FUNCTION_BLOCK FB_TM1K2
(*
    Function block for Arrival Time Monitor (ATM) controls:
    - X, Y motion
    - Y target states
    - thermocouple

    For TM1K2, we make the following adjustments:
    - Add stTarget6 to the inputs
    - Change the array pragma from 1..6 to 1..7 (1 out and 6 in states, up from 5 in states)
    - Use E_TM1K2_States instead of E_ATM_States
	
	Add array to 1..9
*)
VAR_IN_OUT
    // Y motor (state select).
    stYStage: ST_MotionStage;
    // X motor (align target to beam).
    stXStage: ST_MotionStage;
    // The fast fault output to fault to.
    fbFFHWO: FB_HardwareFFOutput;
    // The arbiter to request beam conditions from.
    fbArbiter: FB_Arbiter;
END_VAR
VAR_INPUT
    // Settings for the OUT state.
    stOut: ST_PositionState;
    // Settings for the TARGET1 state.
    stTarget1: ST_PositionState;
    // Settings for the TARGET2 state.
    stTarget2: ST_PositionState;
    // Settings for the TARGET3 state.
    stTarget3: ST_PositionState;
    // Settings for the TARGET4 state.
    stTarget4: ST_PositionState;
    // Settings for the TARGET5 state.
    stTarget5: ST_PositionState;
    // Settings for the TARGET6 state.
    stTarget6: ST_PositionState;
    // Settings for the TARGET7 state.
    stTarget7: ST_PositionState;
    // Settings for the TARGET8 state.
    stTarget8: ST_PositionState;
    // Set this to a non-unknown value to request a new move.
    {attribute 'pytmc' := '
        pv: MMS:STATE:SET
        io: io
    '}
    eEnumSet: E_TM1K2_States;
    // Set this to TRUE to enable input state moves, or FALSE to disable them.
    bEnableMotion: BOOL;
    // Set this to TRUE to enable beam parameter checks, or FALSE to disable them.
    bEnableBeamParams: BOOL;
    // Set this to TRUE to enable position limit checks, or FALSE to disable them.
    bEnablePositionLimits: BOOL;
    // The name of the device for use in the PMPS DB lookup and diagnostic screens.
    sDeviceName: STRING;
    // The name of the transition state in the PMPS database.
    sTransitionKey: STRING;
    // Set this to TRUE to re-read the loaded database immediately (useful for debug).
    bReadDBNow: BOOL;
END_VAR
VAR_OUTPUT
    // The current position state as an enum.
    {attribute 'pytmc' := '
        pv: MMS:STATE:GET
        io: i
    '}
    eEnumGet: E_TM1K2_States;
    // The PMPS database lookup associated with the current position state.
    stDbStateParams: ST_DbStateParams;
END_VAR
VAR
    bInit: BOOL;

    fbYStage: FB_MotionStage;
    fbXStage: FB_MotionStage;

    fbStateDefaults: FB_PositionState_Defaults;

    {attribute 'pytmc' := '
        pv: MMS
        astPositionState.array: 1..7
    '}
    fbStates: FB_PositionStatePMPS1D;
    astPositionState: ARRAY[1..GeneralConstants.MAX_STATES] OF ST_PositionState;
    fbArrCheckWrite: FB_CheckPositionStateWrite;

    {attribute 'pytmc' := 'pv: STC:01'}
    fbThermoCouple1: FB_TempSensor;

    {attribute 'pytmc' :='pv: FWM'}
    fbFlowMeter: FB_AnalogInput := (iTermBits:=15, fTermMax:=60, fTermMin:=0);
END_VAR
VAR CONSTANT
    // State defaults if not provided
    fDelta: LREAL := 2;
    fAccel: LREAL := 200;
    fOutDecel: LREAL := 25;
END_VAR


IF NOT bInit THEN
    bInit := TRUE;

    stYStage.nEnableMode := E_StageEnableMode.DURING_MOTION;
    stXStage.nEnableMode := E_StageEnableMode.DURING_MOTION;

    // Partial backcompat, this used to set fVelocity too but this should be set per install
    fbStateDefaults(stPositionState:=stOut, sNameDefault:='OUT', fDeltaDefault:=fDelta, fAccelDefault:=fAccel, fDecelDefault:=fOutDecel);
    fbStateDefaults(stPositionState:=stTarget1, sNameDefault:='TARGET1', fDeltaDefault:=fDelta, fAccelDefault:=fAccel, fDecelDefault:=fAccel);
    fbStateDefaults(stPositionState:=stTarget2, sNameDefault:='TARGET2', fDeltaDefault:=fDelta, fAccelDefault:=fAccel, fDecelDefault:=fAccel);
    fbStateDefaults(stPositionState:=stTarget3, sNameDefault:='TARGET3', fDeltaDefault:=fDelta, fAccelDefault:=fAccel, fDecelDefault:=fAccel);
    fbStateDefaults(stPositionState:=stTarget4, sNameDefault:='TARGET4', fDeltaDefault:=fDelta, fAccelDefault:=fAccel, fDecelDefault:=fAccel);
    fbStateDefaults(stPositionState:=stTarget5, sNameDefault:='TARGET5', fDeltaDefault:=fDelta, fAccelDefault:=fAccel, fDecelDefault:=fAccel);
    fbStateDefaults(stPositionState:=stTarget6, sNameDefault:='TARGET6', fDeltaDefault:=fDelta, fAccelDefault:=fAccel, fDecelDefault:=fAccel);
    fbStateDefaults(stPositionState:=stTarget7, sNameDefault:='TARGET7', fDeltaDefault:=fDelta, fAccelDefault:=fAccel, fDecelDefault:=fAccel);
    fbStateDefaults(stPositionState:=stTarget8, sNameDefault:='TARGET8', fDeltaDefault:=fDelta, fAccelDefault:=fAccel, fDecelDefault:=fAccel);
END_IF

stYStage.bHardwareEnable := TRUE;
stYStage.bPowerSelf := FALSE;

stXStage.bLimitForwardEnable := TRUE;
stXStage.bLimitBackwardEnable := TRUE;
stXStage.bHardwareEnable := TRUE;
stXStage.bPowerSelf := TRUE;

fbYStage(stMotionStage:=stYStage);
fbXStage(stMotionStage:=stXStage);

// We need to update from PLC or from EPICS, but not both
fbArrCheckWrite(
    astPositionState:=astPositionState,
    bCheck:=TRUE,
    bSave:=FALSE,
);
IF NOT fbArrCheckWrite.bHadWrite THEN
    astPositionState[E_TM1K2_States.OUT] := stOut;
    astPositionState[E_TM1K2_States.TARGET1] := stTarget1;
    astPositionState[E_TM1K2_States.TARGET2] := stTarget2;
    astPositionState[E_TM1K2_States.TARGET3] := stTarget3;
    astPositionState[E_TM1K2_States.TARGET4] := stTarget4;
    astPositionState[E_TM1K2_States.TARGET5] := stTarget5;
    astPositionState[E_TM1K2_States.TARGET6] := stTarget6;
    astPositionState[E_TM1K2_States.TARGET7] := stTarget7;
    astPositionState[E_TM1K2_States.TARGET8] := stTarget8;
END_IF

fbStates(
    stMotionStage:=stYStage,
    astPositionState:=astPositionState,
    eEnumSet:=eEnumSet,
    eEnumGet:=eEnumGet,
    fbFFHWO:=fbFFHWO,
    fbArbiter:=fbArbiter,
    bEnableMotion:=bEnableMotion,
    bEnableBeamParams:=bEnableBeamParams,
    bEnablePositionLimits:=bEnablePositionLimits,
    sDeviceName:=sDeviceName,
    sTransitionKey:=sTransitionKey,
    bReadDBNow:=bReadDBNow,
    stDbStateParams=>stDbStateParams,
);

fbArrCheckWrite(
    astPositionState:=astPositionState,
    bCheck:=FALSE,
    bSave:=TRUE,
);

stOut := astPositionState[E_TM1K2_States.OUT];
stTarget1 := astPositionState[E_TM1K2_States.TARGET1];
stTarget2 := astPositionState[E_TM1K2_States.TARGET2];
stTarget3 := astPositionState[E_TM1K2_States.TARGET3];
stTarget4 := astPositionState[E_TM1K2_States.TARGET4];
stTarget5 := astPositionState[E_TM1K2_States.TARGET5];
stTarget6 := astPositionState[E_TM1K2_States.TARGET6];
stTarget7 := astPositionState[E_TM1K2_States.TARGET7];
stTarget8 := astPositionState[E_TM1K2_States.TARGET8];

fbThermoCouple1();
fbFlowMeter();

END_FUNCTION_BLOCK

(* stored: Version 1.1.0.1, ProductVersion 3.1.4024.12
   POU FB_TM1K2: Id {7f8d0764-a8fd-47be-89c9-262437998617}, SpecialFunc None *)
